// TIA Portal V18 export
FUNCTION_BLOCK "Simulation"   // FB6, FBD
TITLE = Simulation
{ S7_Optimized_Access := 'TRUE' }
VERSION : 0.1
// Simulates machine behavior
// stored: AutoNumber true, IsIECCheckEnabled true, IsRetainMemResEnabled false, MemoryReserve 100, SetENOAutomatically false, UDAEnableTagReadback false
   VAR_INPUT
      moveUp : Bool;
      moveDown : Bool;
      moveLeft : Bool;
      moveRight : Bool;
      runConveyor : Bool;
      engineBroken : Bool;
      robotGoToStation : Bool;
      robotGoToMagazine : Bool;
   END_VAR
   VAR_OUTPUT
      xPosition : Int;
      yPosition : Int;
      lightBeam1 : Bool;
      lightBeam2 : Bool;
      lightBeam3 : Bool;
      robotPosHMI : Int;
      robotHasChip : Bool;
   END_VAR
   VAR
      instTimerSimulate { S7_SetPoint := 'True'} : TON_TIME;
      statSimulate : Bool;
      statPositionConveyor : Int;
      statRobotHasChip : Bool;
      statRobotPosHMI : Int;
   END_VAR
   VAR_TEMP
      tempLB1 : Bool;
      tempLB2 : Bool;
      tempLB3 : Bool;
   END_VAR
   VAR CONSTANT
      SIMULATION_TIME : Time := T#10ms;
   END_VAR
BEGIN

REGION Network 1 (SCL)
   //=============================================================================
   //Siemens AG // (c)Copyright (2018)
   //-----------------------------------------------------------------------------
   // Library: -
   // Tested with: CPU 1517-3 PN/DP V2.5
   // Engineering: TIA Portal V15
   // Restrictions: -
   // Requirements: PLC (S7-1500)
   // Functionality: Simulation
   //-----------------------------------------------------------------------------
   // Change log table:
   // Version  Date      Expert in charge  Changes applied
   // 01.00.00 24.08.18  Siemens           First released version
   //=============================================================================
END_REGION

REGION Network 2: trigger simulation step
   // set bit for one cycle every 10ms
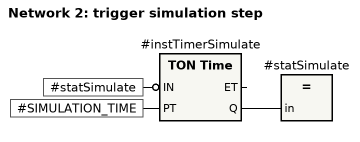
   #instTimerSimulate(IN := NOT #statSimulate, PT := #SIMULATION_TIME);   // TON
   #statSimulate := #instTimerSimulate.Q;
END_REGION

REGION Network 3 (SCL): simulation step
   //=============================================================================
   //Siemens AG // (c)Copyright (2018)
   //-----------------------------------------------------------------------------
   // Library: (that the source is dedicated to)
   // Tested with: (test system with FW version)
   // Engineering: TIA Portal V15
   // Restrictions: (OB types, etc.)
   // Requirements: (hardware, technological package, memory needed, etc.)
   // Functionality: (that is implemented in the block)
   //-----------------------------------------------------------------------------
   // Change log table:
   // Version Date Expert in charge Changes applied
   // 24.08.18 dd.mm.yyyy (Name of expert) First released version
   //=============================================================================


   IF (#statSimulate = TRUE)
     AND (NOT #engineBroken)
   THEN
     //move robot
     IF (#moveUp = TRUE)
     THEN
       #yPosition += 1;
     END_IF;
     IF (#moveDown = TRUE)
     THEN
       #yPosition -= 1;
     END_IF;
     IF (#moveLeft = TRUE)
     THEN
       #xPosition += 1;
     END_IF;
     IF (#moveRight = TRUE)
     THEN
       #xPosition -= 1;
     END_IF;
     //move conveyor
     IF (#statPositionConveyor > 800)
     THEN
       #statPositionConveyor := 0;
     ELSIF (#runConveyor = TRUE)
     THEN
       #statPositionConveyor += 1;
     END_IF;
   END_IF;

   //for S7-300 / S7-400
   #tempLB1 := FALSE;
   #tempLB2 := FALSE;
   #tempLB3 := FALSE;

   //assign lightbeams
   CASE #statPositionConveyor OF
     30..60:
       #tempLB1 := TRUE;
     500..530:
       #tempLB2 := TRUE;
     780..800:
       #tempLB3 := TRUE;

     ELSE  // Statement section ELSE
       ;
   END_CASE;

   #lightBeam1 := #tempLB1;
   #lightBeam2 := #tempLB2;
   #lightBeam3 := #tempLB3;

   //Calculate data for display of robot in HMI
   IF (#xPosition = 100)
   THEN
     #statRobotPosHMI := #yPosition;
   ELSE
       #statRobotPosHMI :=100;
   END_IF;

   IF (#robotGoToStation)
   THEN
       #statRobotHasChip := TRUE;
   END_IF;
   IF (#robotGoToMagazine = TRUE)
     OR (#statRobotPosHMI = 0)
   THEN
     #statRobotHasChip := FALSE;
   END_IF;

   // wirte outputs
   #robotHasChip:= #statRobotHasChip;
   #robotPosHMI := #statRobotPosHMI;
END_REGION
END_FUNCTION_BLOCK
